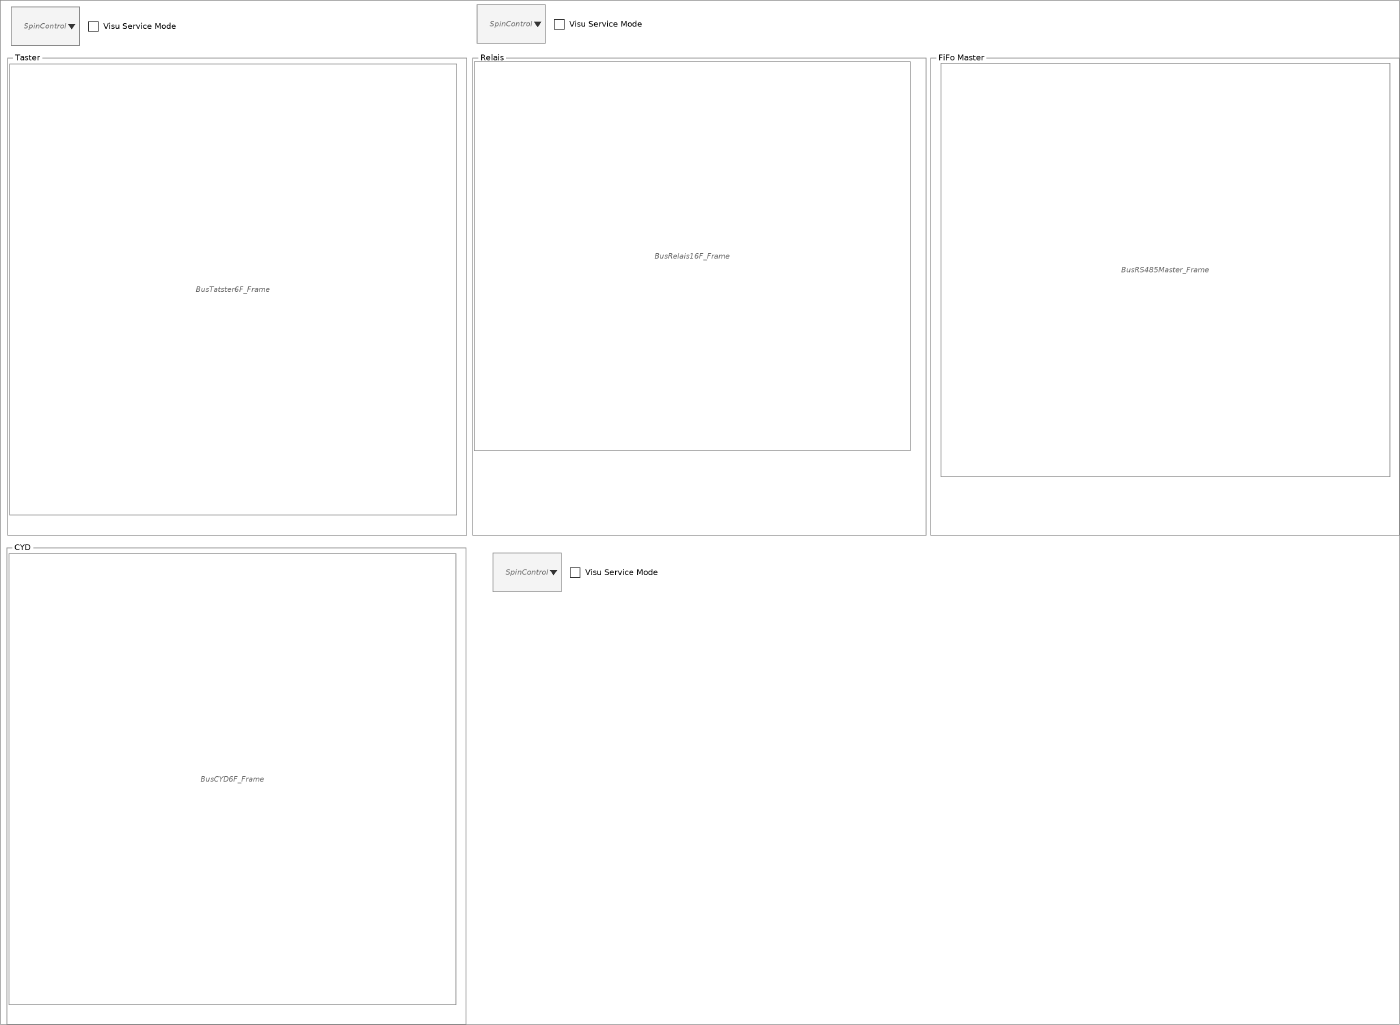
VISUALIZATION RS485HB_ServiceVISU_1  // 1938x1419
    SpinControl (15,9 95x54), variable: GVL_ServiceVisu.iDeviceTasterVisu
        p651134158: cMaxBusTaster
    Checkbox (120,7 181x59), "Visu Service Mode", variable: GVL_ServiceVisu.bTasterServiceAktiv[GVL_ServiceVisu.iDeviceTasterVisu]
    SpinControl (660,6 95x54), variable: GVL_ServiceVisu.iDeviceRelaisVisu
        p576042468: cMaxBusTaster+1
        p651134158: cMaxBusRelais +cMaxBusTaster +1
    Checkbox (765,4 181x59), "Visu Service Mode", variable: GVL_ServiceVisu.bRelaisServiceAktiv[GVL_ServiceVisu.iDeviceRelaisVisu]
    GroupBox (654,72 628x669), "Relais"
        Frame (2,13 604x539)
            shows BusRelais16F_Frame(ST_BusRelais16F_Input := GVL_ServiceVisu.stRelaisService[GVL_ServiceVisu.iDeviceRelaisVisu], ST_BusRelais16F_Output := fbRelaisHB16F[GVL_ServiceVisu.iDeviceRelaisVisu].Q_stOutput, ST_BusRelais16F_Cnt := fbRelaisHB16F[GVL_ServiceVisu.iDeviceRelaisVisu].Q_stCnt)
    GroupBox (10,72 636x669), "Taster"
        Frame (3,16 619x625)
            shows BusTatster6F_Frame(stBusTaster6F_Input := GVL_ServiceVisu.stTasterService[GVL_ServiceVisu.iDeviceTasterVisu], stBusTaster6F_Output := fbTasterHB6F[GVL_ServiceVisu.iDeviceTasterVisu].Q_stOutput, stBusTaster6F_Cnt := fbTasterHB6F[GVL_ServiceVisu.iDeviceTasterVisu].Q_stCnt)
    GroupBox (1288,72 650x669), "FiFo Master"
        Frame (14,15 622x573)
            shows BusRS485Master_Frame(bBusBelastungstest := RS485_COM_PRG.fbRS485SendCmdFiFo.I_bBusBelastungstest, bReset := RS485_COM_PRG.fbRS485SendCmdFiFo.I_bReset, stFiFoMasterState := RS485_COM_PRG.fbRS485SendCmdFiFo.Q_stStates, stRS48StartupState := RS485_COM_PRG.fbRS485Startup.Q_stStates)
            shows BusRS485Master_Frame()
    GroupBox (9,750 636x669), "CYD"
        Frame (3,16 619x625)
            shows BusCYD6F_Frame(stBusTaster6F_Input := GVL_ServiceVisu.stCYDService[GVL_ServiceVisu.iDeviceCYDVisu], stBusTaster6F_Output := fbCYDHB6F[GVL_ServiceVisu.iDeviceCYDVisu].Q_stOutput, stBusTaster6F_Cnt := fbCYDHB6F[GVL_ServiceVisu.iDeviceCYDVisu].Q_stCnt)
    SpinControl (682,765 95x54), variable: GVL_ServiceVisu.iDeviceCYDVisu
        p576042468: cMaxBusRelais +cMaxBusTaster +2
        p651134158: cMaxCYD+cMaxBusRelais +cMaxBusTaster +1
    Checkbox (787,763 181x59), "Visu Service Mode", variable: GVL_ServiceVisu.bCYDServiceAktiv[GVL_ServiceVisu.iDeviceCYDVisu]
END_VISUALIZATION

(* stored: Version 1.1.0.1, ProductVersion 3.1.4024.12
   Visu RS485HB_ServiceVISU_1: Id {06c39a48-d174-49d6-8ee8-1ee083b6bb1f} *)
